{attribute 'qualified_only'}
VAR_GLOBAL CONSTANT
	LIST_SIZE : UINT := 100; // Number of list items.
END_VAR

(* stored: Version 1.1.0.1, ProductVersion 3.1.4020.12
   GVL GVL_List: Id {9b47b2a7-38a5-4620-aafc-3dbeb164f5d3}, ParameterList True *)
